# EPICS StreamDevice protocol: aeroflexSup/aeroflex_2030.proto
InTerminator = '\n';
OutTerminator = '\n';

getCarrierFrequency {
	out "cfrq?";
	in ":CFRQ:VALUE %f;INC %*f";
}

getModulation {
	out "mode?";
	in ":MODE %{AM,FM|AM,PM|AM|FM,PULSE|FM|PM,PULSE|PM}";
}

setModulation {
	out "MODE %{AM,FM|AM,PM|AM|FM,PULSE|FM|PM,PULSE|PM}";
}
